(* IEC 61131-3 sources: repolevel_ST_code_completion/output/full_case_fixed/repoeval_ProductionLine/readful_result_history, 20 files *)

(* ---- Motor_0.st ---- *)
FUNCTION_BLOCK Motor
VAR_INPUT
	MotorI:MotorI;
END_VAR
VAR_OUTPUT
	MotorO:MotorO;
END_VAR
VAR
	WaitTimer: TON;
	InternalSequenceDelay: TIME;
END_VAR

IF MotorI.Overload THEN
	MotorO.FaultStatus := TRUE;
	MotorO.Coil := FALSE;
	RETURN;
END_IF

IF MotorO.FaultStatus = FALSE THEN
	WaitTimer(IN := TRUE, PT := InternalSequenceDelay);
END_IF

IF WaitTimer.Q THEN
	MotorO.Coil := TRUE;
	WaitTimer(IN := FALSE);
END_IF

RETURN;
END_FUNCTION_BLOCK

(* ---- Motor_1.st ---- *)
FUNCTION_BLOCK Motor
VAR_INPUT
	MotorI:MotorI;
END_VAR
VAR_OUTPUT
	MotorO:MotorO;
END_VAR
VAR
	WaitTimer: TON;
	InternalSequenceDelay: TIME;
END_VAR

IF MotorI.Overload THEN
	MotorO.FaultStatus := TRUE;
	MotorO.Coil := FALSE;
	RETURN;
END_IF

IF MotorO.FaultStatus = FALSE THEN
WaitTimer.IN := TRUE; // Setting the 'IN' input for the TON block instance.
  WaitTimer.PT := InternalSequenceDelay; // Setting the 'PT' (preset time) input for the TON block instance.
  WaitTimer(); // Executing the TON instance.
END_IF

IF WaitTimer.Q THEN
	MotorO.Coil := TRUE;
WaitTimer.IN := FALSE; // Resetting the 'IN' input for the TON block instance.
  WaitTimer(); // Executing the TON instance to ensure state updates.
END_IF

RETURN;
END_FUNCTION_BLOCK

(* ---- Motor_2.st ---- *)
FUNCTION_BLOCK Motor
VAR_INPUT
	MotorI:MotorI;
END_VAR
VAR_OUTPUT
	MotorO:MotorO;
END_VAR
VAR
	WaitTimer: TON;
	InternalSequenceDelay: TIME;
END_VAR

IF MotorI.Overload THEN
	MotorO.FaultStatus := TRUE;
	MotorO.Coil := FALSE;
	RETURN;
END_IF

IF MotorO.FaultStatus = FALSE THEN
WaitTimer.IN := TRUE; // Setting the 'IN' input for the TON block instance.
  WaitTimer.PT := InternalSequenceDelay; // Setting the 'PT' (preset time) input for the TON block instance.
  WaitTimer(); // Executing the TON instance.
END_IF

IF WaitTimer.Q THEN
	MotorO.Coil := TRUE;
WaitTimer.IN := FALSE; // Resetting the 'IN' input for the TON block instance.
  WaitTimer(); // Executing the TON instance to ensure state updates.
END_IF

RETURN;
END_FUNCTION_BLOCK

(* ---- Motor_3.st ---- *)
FUNCTION_BLOCK Motor
VAR_INPUT
	MotorI:MotorI;
END_VAR
VAR_OUTPUT
	MotorO:MotorO;
END_VAR
VAR
	WaitTimer: TON;
	InternalSequenceDelay: TIME;
END_VAR

IF MotorI.Overload THEN
	MotorO.FaultStatus := TRUE;
	MotorO.Coil := FALSE;
	RETURN;
END_IF

IF MotorO.FaultStatus = FALSE THEN
WaitTimer.IN := TRUE; // Setting the 'IN' input for the TON block instance.
  WaitTimer.PT := InternalSequenceDelay; // Setting the 'PT' (preset time) input for the TON block instance.
  WaitTimer(); // Executing the TON instance.
END_IF

IF WaitTimer.Q THEN
	MotorO.Coil := TRUE;
WaitTimer.IN := FALSE; // Resetting the 'IN' input for the TON block instance.
  WaitTimer(); // Executing the TON instance to ensure state updates.
END_IF

RETURN;
END_FUNCTION_BLOCK

(* ---- Motor_ResetFault_0.st ---- *)
METHOD ResetFault : BOOL
VAR_INPUT
	MotorI:MotorI;
END_VAR
VAR_OUTPUT
	MotorO:MotorO;
END_VAR
VAR
	ResetDetect: r_trig;
END_VAR

ResetDetect(CLK := MotorI.FaultReset);

IF ResetDetect.Q THEN
	MotorO.FaultStatus := FALSE;
END_IF
END_OTHER

(* ---- Motor_ResetFault_1.st ---- *)
METHOD ResetFault : BOOL
VAR_INPUT
  MotorI:MotorI;
END_VAR
VAR_OUTPUT
  MotorO:MotorO;
END_VAR
VAR
  ResetDetect: r_trig;
END_VAR

ResetDetect(CLK := MotorI.FaultReset);

IF ResetDetect.Q THEN
  MotorO.FaultStatus := FALSE;
END_IF
END_METHOD

(* ---- Motor_SetFault_0.st ---- *)
METHOD SetFault : BOOL
VAR_INPUT
	MotorI:MotorI;
END_VAR
VAR_OUTPUT
	MotorO:MotorO;
END_VAR
VAR
	WaitTimer:TON;
	InternalSequenceDelay:TIME;
END_VAR

IF MotorI.Overload THEN
	MotorO.FaultStatus := TRUE;
	MotorO.Coil := FALSE;
END_IF
END_OTHER

(* ---- Motor_SetFault_1.st ---- *)
METHOD SetFault : BOOL
VAR_INPUT
  MotorI:MotorI;
END_VAR
VAR_OUTPUT
  MotorO:MotorO;
END_VAR
VAR
  WaitTimer:TON;
  InternalSequenceDelay:TIME;
END_VAR

IF MotorI.Overload THEN
  MotorO.FaultStatus := TRUE;
  MotorO.Coil := FALSE;
END_IF

(* ---- Motor_SetWaitTime_0.st ---- *)
METHOD SetWaitTime : BOOL
VAR_INPUT
	MotorI:MotorI;
	SequenceDelay:TIME;
END_VAR
VAR_OUTPUT
	MotorO:MotorO;
END_VAR
VAR
	WaitTimer:TON;
	InternalSequenceDelay:TIME;
END_VAR

InternalSequenceDelay := SequenceDelay;

IF MotorO.FaultStatus = FALSE THEN
	WaitTimer(IN := TRUE, PT := InternalSequenceDelay);
END_IF

IF WaitTimer.Q THEN
	MotorO.Coil := TRUE;
	WaitTimer(IN := FALSE);
END_IF

RETURN;
END_OTHER

(* ---- Motor_SetWaitTime_1.st ---- *)
METHOD SetWaitTime : BOOL
VAR_INPUT
  MotorI:MotorI;
  SequenceDelay:TIME;
END_VAR
VAR_OUTPUT
  MotorO:MotorO;
END_VAR
VAR
  WaitTimer:TON;
  InternalSequenceDelay:TIME;
END_VAR

InternalSequenceDelay := SequenceDelay;

IF MotorO.FaultStatus = FALSE THEN
  // Start the timer when there is no fault
  WaitTimer(IN := TRUE, PT := InternalSequenceDelay);
END_IF

IF WaitTimer.Q THEN
  // Activate MotorO coil when WaitTimer indicates timeout
  MotorO.Coil := TRUE;
  // Reset the timer
  WaitTimer(IN := FALSE);
END_IF

RETURN;
// Replace incorrect keyword "END_OTHER" with "END_METHOD"
END_METHOD

(* ---- Motor_SetWaitTime_2.st ---- *)
METHOD SetWaitTime : BOOL
VAR_INPUT
 MotorI:MotorI;
 SequenceDelay:TIME;
END_VAR
VAR_OUTPUT
 MotorO:MotorO;
END_VAR
VAR
 WaitTimer:TON;
 InternalSequenceDelay:TIME;
END_VAR

InternalSequenceDelay := SequenceDelay;

IF MotorO.FaultStatus = FALSE THEN
 // Start the timer when there is no fault
 WaitTimer(IN := TRUE, PT := InternalSequenceDelay);
END_IF

IF WaitTimer.Q THEN
 // Activate MotorO coil when WaitTimer indicates timeout
 MotorO.Coil := TRUE;
 // Stop the timer by setting IN to FALSE only if it's still running
 IF WaitTimer.IN THEN
  WaitTimer(IN := FALSE);
 END_IF
END_IF

RETURN;
// Replace incorrect keyword "END_OTHER" with "END_METHOD"
END_METHOD

(* ---- Motor_SetWaitTime_3.st ---- *)
METHOD SetWaitTime : BOOL
VAR_INPUT
MotorI:MotorI;
SequenceDelay:TIME;
END_VAR
VAR_OUTPUT
MotorO:MotorO;
END_VAR
VAR
WaitTimer:TON;
InternalSequenceDelay:TIME;
END_VAR

InternalSequenceDelay := SequenceDelay;

IF MotorO.FaultStatus = FALSE THEN
// Start the timer when there is no fault
WaitTimer(IN := TRUE, PT := InternalSequenceDelay); // Correctly call TON instance
END_IF

IF WaitTimer.Q THEN
// Activate MotorO coil when WaitTimer indicates timeout
MotorO.Coil := TRUE;
// Stop the timer; no need to check "WaitTimer.IN" explicitly
WaitTimer(IN := FALSE); // Correctly call TON instance again to reset it
END_IF

RETURN;
// Replace incorrect keyword "END_OTHER" with "END_METHOD"
END_METHOD

(* ---- Motor_TurnOff_0.st ---- *)
METHOD TurnOff : BOOL
VAR_INPUT
	MotorI:MotorI;
END_VAR
VAR_OUTPUT
	MotorO:MotorO;
END_VAR
VAR
	WaitTimer:TON;
	InternalSequenceDelay:TIME;
END_VAR

MotorO.Coil := FALSE;
RETURN;
END_OTHER

(* ---- Motor_TurnOff_1.st ---- *)
METHOD TurnOff : BOOL
VAR_INPUT
	MotorI:MotorI;
END_VAR
VAR_OUTPUT
	MotorO:MotorO;
END_VAR
VAR
	WaitTimer:TON;
	InternalSequenceDelay:TIME;
END_VAR

MotorO.Coil := FALSE;
RETURN;
END_OTHER

(* ---- Motor_TurnOff_2.st ---- *)
METHOD TurnOff : BOOL
VAR_INPUT
	MotorI:MotorI;
END_VAR
VAR_OUTPUT
	MotorO:MotorO;
END_VAR
VAR
	WaitTimer:TON;
	InternalSequenceDelay:TIME;
END_VAR

MotorO.Coil := FALSE;
RETURN;
END_OTHER

(* ---- Motor_TurnOff_3.st ---- *)
METHOD TurnOff : BOOL
VAR_INPUT
	MotorI:MotorI;
END_VAR
VAR_OUTPUT
	MotorO:MotorO;
END_VAR
VAR
	WaitTimer:TON;
	InternalSequenceDelay:TIME;
END_VAR

MotorO.Coil := FALSE;
RETURN;
END_OTHER

(* ---- Motor_TurnOn_0.st ---- *)
METHOD TurnOn : BOOL
VAR_INPUT
	MotorI:MotorI;
END_VAR
VAR_OUTPUT
	MotorO:MotorO;
END_VAR
VAR
	WaitTimer:TON;
	InternalSequenceDelay:TIME;
END_VAR

IF MotorO.FaultStatus = FALSE THEN
	WaitTimer(IN := TRUE, PT := InternalSequenceDelay);
END_IF

IF WaitTimer.Q THEN
	MotorO.Coil := TRUE;
	WaitTimer(IN := FALSE);
END_IF

RETURN;
END_OTHER

(* ---- Motor_TurnOn_1.st ---- *)
METHOD TurnOn : BOOL
VAR_INPUT
  MotorI:MotorI;
END_VAR
VAR_OUTPUT
  MotorO:MotorO;
END_VAR
VAR
  WaitTimer:TON;
  InternalSequenceDelay:TIME;
END_VAR

IF MotorO.FaultStatus = FALSE THEN
  WaitTimer.IN := TRUE; // Correctly set the IN property
  WaitTimer.PT := InternalSequenceDelay; // Assign PT if needed
END_IF

IF WaitTimer.Q THEN
  MotorO.Coil := TRUE;
  WaitTimer.IN := FALSE; // Properly reset the IN property
END_IF

RETURN;
END_METHOD // Correct termination of METHOD

(* ---- Motor_TurnOn_2.st ---- *)
METHOD TurnOn : BOOL
VAR_INPUT
 MotorI:MotorI;
END_VAR
VAR_OUTPUT
 MotorO:MotorO;
END_VAR
VAR
 WaitTimer:TON;
 InternalSequenceDelay:TIME;
END_VAR

IF MotorO.FaultStatus = FALSE THEN
 WaitTimer.IN := TRUE;
 WaitTimer.PT := InternalSequenceDelay;
 WaitTimer(); // Execute the TON function block
END_IF

IF WaitTimer.Q THEN
 MotorO.Coil := TRUE;
 WaitTimer.IN := FALSE;
 WaitTimer(); // Execute the TON function block after modifying IN
END_IF

RETURN;
END_METHOD

(* ---- Motor_TurnOn_3.st ---- *)
METHOD TurnOn : BOOL
VAR_INPUT
MotorI:MotorI;
END_VAR
VAR_OUTPUT
MotorO:MotorO;
END_VAR
VAR
WaitTimer:TON;
InternalSequenceDelay:TIME;
END_VAR

// Ensure WaitTimer executes only when necessary
IF MotorO.FaultStatus = FALSE THEN
WaitTimer.IN := TRUE;
WaitTimer.PT := InternalSequenceDelay;
WaitTimer(); // Execute the TON function block
END_IF

IF WaitTimer.Q THEN
MotorO.Coil := TRUE;

// Reset the timer only if necessary
IF WaitTimer.IN THEN
 WaitTimer.IN := FALSE;
 WaitTimer(); // Call TON to reflect the reset state
END_IF
END_IF

RETURN;
END_METHOD
